FUNCTION_BLOCK E_TO_EI (* Convert a Event to a EInit *)
  (* Standard: 61499-2; Description: Copyright (c) 2025 HR Agrartechnik GmbH This program and the accompanying materials are made available under the terms of the Eclipse Public License 2.0 which is available at https://www.eclipse.org/legal/epl-2.0/ SPDX-License-Identifier: EPL-2.0 *)
  (* Version 1.0, 2025-01-21, Franz Höpfinger, HR Agrartechnik GmbH *)
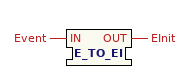
  EVENT_INPUT
    IN; (* Event IN *)
  END_EVENT
  EVENT_OUTPUT
    OUT : EInit; (* EInit OUT *)
  END_EVENT
END_FUNCTION_BLOCK
